{attribute 'qualified_only'}
{attribute 'strict'}
{attribute 'to_string'}
TYPE E_MotionLogLevel :
(
	WARNING := 0,
	ERROR := 1,
	INFO := 2
);
END_TYPE

(* stored: Version 1.1.0.1
   DUT E_MotionLogLevel: Id {17a29375-617a-41ff-83a3-272050e9cb35} *)
